(* IEC 61131-3 sources: ATCMcontrol_Engineering/src/COM/softing/fc/CL/Libs/ATCM_IEC1131_3/table_23, 11 files *)

(* ---- abs.st ---- *)
(*[[
    UserURL= "ATCMFile:ABS.htm"
]]*)

FUNCTION ABS : ANY_NUM
VAR_INPUT
    IN : ANY_NUM;
END_VAR

overload () inline{java.lang.Math.abs(%1)}

END_FUNCTION

(* ---- acos.st ---- *)
(*[[
    UserURL= "ATCMFile:ACOS.htm"
]]*)
FUNCTION ACOS : ANY_REAL
VAR_INPUT
    IN : ANY_REAL;
END_VAR

overload () inline{java.lang.Math.acos(%1)}

END_FUNCTION

(* ---- asin.st ---- *)
(*[[
    UserURL= "ATCMFile:ASIN.htm"
]]*)

FUNCTION ASIN : ANY_REAL
VAR_INPUT
    IN : ANY_REAL;
END_VAR

overload () inline{java.lang.Math.asin(%1)}

END_FUNCTION

(* ---- atan.st ---- *)
(*[[
    UserURL= "ATCMFile:ATAN.htm"
]]*)

FUNCTION ATAN : ANY_REAL
VAR_INPUT
    IN : ANY_REAL;
END_VAR

overload () inline{java.lang.Math.atan(%1)}

END_FUNCTION

(* ---- cos.st ---- *)
(*[[
    UserURL= "ATCMFile:COS.htm"
]]*)

FUNCTION COS : ANY_REAL
VAR_INPUT
    IN : ANY_REAL;
END_VAR

overload () inline{java.lang.Math.cos(%1)}

END_FUNCTION

(* ---- exp.st ---- *)
(*[[
    UserURL= "ATCMFile:EXP.htm"
]]*)

FUNCTION EXP : ANY_REAL
VAR_INPUT
    IN : ANY_REAL;
END_VAR

overload () inline{java.lang.Math.exp(%1)}

END_FUNCTION

(* ---- ln.st ---- *)
(*[[
    UserURL= "ATCMFile:LN.htm"
]]*)

FUNCTION LN : ANY_REAL
VAR_INPUT
    IN : ANY_REAL;
END_VAR

overload () inline{java.lang.Math.log(%1)}

END_FUNCTION

(* ---- log.st ---- *)
(*[[
    UserURL= "ATCMFile:LOG.htm"
]]*)

FUNCTION LOG : ANY_REAL
VAR_INPUT
    IN : ANY_REAL;
END_VAR

overload () inline{java.lang.Math.log(%1)/java.lang.Math.log(10)}

END_FUNCTION

(* ---- sin.st ---- *)
(*[[
    UserURL= "ATCMFile:SIN.htm"
]]*)

FUNCTION SIN : ANY_REAL
VAR_INPUT
    IN : ANY_REAL;
END_VAR

overload () inline{java.lang.Math.sin(%1)}

END_FUNCTION

(* ---- sqrt.st ---- *)
(*[[
    UserURL= "ATCMFile:SQRT.htm"
]]*)

FUNCTION SQRT : ANY_REAL
VAR_INPUT
    IN : ANY_REAL;
END_VAR

overload () inline{java.lang.Math.sqrt(%1)}

END_FUNCTION

(* ---- tan.st ---- *)
(*[[
    UserURL= "ATCMFile:TAN.htm"
]]*)

FUNCTION TAN : ANY_REAL
VAR_INPUT
    IN : ANY_REAL;
END_VAR

overload () inline{java.lang.Math.tan(%1)}

END_FUNCTION
